PROGRAM Main2
VAR	
	Sequence2 				: Sequence2;
	Reset2					: FB_ResetAllAxis;
	fbStopAll				: FB_StopAll;
	fbPowerAll				: FB_PowerAll;
	bSequenceExecute		: BOOL;
	bUserIncrementStep		: BOOL;
	bUserInfiniteMovement	: BOOL;
	bResetExecute			: BOOL;
	MainState 				: MainStateAxis_enum;
	mainCommands			: MainCommands_typ;
	XYParamaters			: XYParams_typ;
	
	bStopAll: BOOL;
	bPowerEnable: BOOL;
	
	//Test Variables
	
	
	{attribute 'instance-path'}
	{attribute 'no-init'}
	InstancePath			: STRING;
	btest: BOOL;
	AirVariable				AT %Q* : BOOL;
	
	internalEnable			: BOOL;
	internalDisable			: BOOL;
	
	//internalCurrentMoveType	: DeltaCommandType_enum;
	
	internalState			: DeltaState_enum;
	
	internalSetCoordTrafoDone	: BOOL;
	internalMovePathDone		: BOOL;

	
	internalInitObjPos		: ARRAY [1..3] OF MC_LREAL := [0,0,0];
	internalAxesList		: ST_KinAxes;
	internalCMGroup			: AXES_GROUP_REF;
	
	internalTrackAxis		: REFERENCE TO AXIS_REF;
	
	internalPathBuffer		: ARRAY[0..32767] OF BYTE;
	internalPathData		: MC_PATH_DATA_REF( ADR( internalPathBuffer ), SIZEOF( internalPathBuffer ));
		
	externalRoute			: REFERENCE TO Route;	

	internalActiveCoordRef	: MC_COORD_REF;		

	// Internal function blocks
	fbReset_X			: MC_Reset;
	fbReset_Y			: MC_Reset;

	fbPower_X			: MC_Power;
	fbPower_Y			: MC_Power;
	
	fbPower_MCS_X		: MC_Power;
	fbPower_MCS_Y		: MC_Power;
	
	fbAddAxisToGrp			: ARRAY[0..2] OF MC_AddAxisToGroup;
	fbGroupEnable			: MC_GroupEnable;
	
	fbSetCoordTrafo			: MC_SetCoordinateTransform;
	fbMoveLinearPrep		: MC_MoveLinearAbsolutePreparation;
	fbMovePath				: MC_MovePath;
	fbMovePathExt			: MC_MovePath;
	
	//Input Variables
	MotionParameters	: DeltaMotionParameters_typ;			// Motion parameters used by internal motion function blocks	
	myMCSOverride: LREAL := 100.0;
	xSetOverride: BOOL;
	lrGrpOverride: MC_LREAL := 1.0;
	fbMC_GroupSetOverride : MC_GroupSetOverride;
	bTeaching				: BOOL;
	
	//Outputs
	Ready				: BOOL;
	Busy				: BOOL;
	
	Error				: BOOL;
	ErrorID				: UDINT;
	ErrorOrigin			: STRING;
	i: INT;
	
	fbGearIn1:  MC_GearIn;
	bGearIn: BOOL;
END_VAR

(*CASE internalState OF
	DL_IDLE:	// ------------------------------------------------------- idle state
	
		Ready		:= FALSE;
		Busy		:= FALSE;
		
		internalDisable		:= FALSE;
		IF internalEnable THEN
			internalEnable		:= FALSE;
			internalState		:= DL_RESET;
		END_IF
	
	DL_RESET:	// ------------------------------------------------------- resets all axis objects
	
		Ready		:= FALSE;
		Busy		:= TRUE;
		Error		:= FALSE;
		ErrorID		:= 0;
		
		fbReset_X.Execute		:= TRUE;
		fbReset_Y.Execute		:= TRUE;
		
		IF fbReset_X.Done AND
			fbReset_Y.Done THEN
			
			fbReset_X.Execute		:= FALSE;
			fbReset_Y.Execute		:= FALSE;
			
			internalState	:= DL_POWER_AXES;
			
		ELSIF fbReset_X.Error OR
			fbReset_Y.Error THEN
			
			ErrorID; // TODO add whatever the error was for that block
			ErrorOrigin		:= CONCAT( InstancePath, '.fbReset' );
			internalState	:= DL_ERROR; 		
		END_IF
		
	DL_POWER_AXES:	// --------------------------------------------------- energizes all axis objects
	
		Ready		:= FALSE;
		Busy		:= TRUE;
		Error		:= FALSE;
		ErrorID		:= 0;

			fbPower_X.Enable	:= TRUE;
			fbPower_Y.Enable	:= TRUE;

			fbPower_X.Enable_Positive	:= TRUE;
			fbPower_Y.Enable_Positive	:= TRUE;
			
			fbPower_X.Enable_Negative	:= TRUE;
			fbPower_Y.Enable_Negative	:= TRUE;
			
			fbPower_X.Override		:= myMCSOverride;
			fbPower_Y.Override		:= myMCSOverride;
			
			IF fbPower_X.Status AND
				fbPower_Y.Status THEN
				
				internalState	:= DL_ADD_AXES_TO_CM;
				
			ELSIF fbPower_X.Error OR
				fbPower_Y.Error THEN
				
				ErrorID;	// TODO add whatever the error was that block
				ErrorOrigin		:= CONCAT( InstancePath, '.fbPower');
				internalState	:= DL_ERROR;
			END_IF
		
	DL_ADD_AXES_TO_CM:	// ----------------------------------------------- adds MCS axes to CM Group
	
		Ready		:= FALSE;
		Busy		:= TRUE;
		Error		:= FALSE;
		ErrorID		:= 0;

			fbAddAxisToGrp[0].IdentInGroup	:= MCS_X;
			
			fbAddAxisToGrp[1].IdentInGroup	:= MCS_Y;
			
			FOR i := 0 TO 1 DO
				fbAddAxisToGrp[i].Execute		:= TRUE;
			END_FOR
			
			IF fbAddAxisToGrp[0].Done AND
				fbAddAxisToGrp[1].Done THEN
				
				fbAddAxisToGrp[0].Execute	:= FALSE;
				fbAddAxisToGrp[1].Execute	:= FALSE;
				
				internalState	:= DL_ENABLE_CM;
				
			ELSIF fbAddAxisToGrp[0].Error THEN
				fbAddAxisToGrp[0].Execute	:= FALSE;
				fbAddAxisToGrp[1].Execute	:= FALSE;
				
				ErrorID;		// todo : add whichever block errored
				ErrorOrigin		:= CONCAT(InstancePath,'.fbAddAxisToGrp1');
				internalState	:= DL_ERROR;
			ELSIF fbAddAxisToGrp[1].Error THEN
				
				fbAddAxisToGrp[0].Execute	:= FALSE;
				fbAddAxisToGrp[1].Execute	:= FALSE;
				
				ErrorID;		// todo : add whichever block errored
				ErrorOrigin		:= CONCAT(InstancePath,'.fbAddAxisToGrp2');
				internalState	:= DL_ERROR;
			END_IF

	DL_ENABLE_CM:	// ------------------------------------------------------- enables the coordinated motion group
	
		Ready		:= FALSE;
		Busy		:= TRUE;
		Error		:= FALSE;
		ErrorID		:= 0;
		
			fbGroupEnable.Execute		:= TRUE;
			
			IF fbGroupEnable.Done THEN
				internalState	:= DL_RUN;
			ELSIF fbGroupEnable.Error THEN
				ErrorID			:= fbGroupEnable.ErrorId;
				ErrorOrigin		:= CONCAT(InstancePath,'.fbGroupEnable');
				internalState	:= DL_ERROR;
			END_IF
		
	DL_RUN:	// --------------------------------------------------------------- Delta running, ready for commands
	
		Ready		:= TRUE;
		Busy		:= FALSE;
		Error		:= FALSE;
		ErrorID		:= 0;
				
		// reset all commanded function blocks when the execute is recieved
		IF fbSetCoordTrafo.Busy OR fbSetCoordtrafo.CommandAborted THEN
			fbSetCoordTrafo.Execute		:= FALSE;
		ELSIF fbMovePath.Busy OR fbMovePath.CommandAborted THEN
			fbMovePath.Execute			:= FALSE;
		ELSIF fbMovePathEXT.Busy OR fbMovePathEXT.CommandAborted THEN
			fbMovePath.Execute			:= FALSE;
		END_IF
		
		// and catch all internal function block errors
		IF fbSetCoordTrafo.Error THEN
			ErrorID			:= fbSetCoordTrafo.ErrorId;
			ErrorOrigin		:= CONCAT( InstancePath, '.fbSetCoordTrafo' );
			internalState	:= DL_ERROR;
		ELSIF fbMovePath.Error THEN
			ErrorID			:= fbMovePath.ErrorId;
			ErrorOrigin		:= CONCAT( InstancePath, '.fbMovePath' );
			internalState	:= DL_ERROR;
		ELSIF fbMovePathEXT.Error THEN
			ErrorID			:= fbMovePathEXT.ErrorId;
			ErrorOrigin		:= CONCAT( InstancePath, '.fbMovePathEXT' );
			internalState	:= DL_ERROR;
		END_IF
	
	DL_ERROR:	// ----------------------------------------------------------- Error state
	
		Ready		:= FALSE;
		Busy		:= FALSE;
		Error		:= TRUE;
	
END_CASE

fbReset_X( Axis := GVL_XY.stAxis[1] );
fbReset_Y( Axis := GVL_XY.stAxis[2] );

fbPower_X( Axis := GVL_XY.stAxis[1] );
fbPower_Y( Axis := GVL_XY.stAxis[2] );

(*fbPower_MCS_X( Axis := GVL_XY.stAxis[1] );
fbPower_MCS_Y( Axis := GVL_XY.stAxis[2] );*)

fbAddAxisToGrp[0]( AxesGroup := internalCMGroup, Axis := GVL_XY.stAxis[1] );
fbAddAxisToGrp[1]( AxesGroup := internalCMGroup, Axis := GVL_XY.stAxis[2] );

fbGroupEnable( AxesGroup := internalCMGroup );

fbSetCoordTrafo( AxesGroup := internalCMGroup );

fbMovePath( AxesGroup := internalCMGroup, PathData := internalPathData );
fbMovePathEXT( AxesGroup := internalCMGroup, PathData := externalRoute.PathData );

fbMC_GroupSetOverride(
	AxesGroup:= internalCMGroup, 
	Enable:= xSetOverride, 
	VelFactor:= lrGrpOverride, 
	Enabled=> , 
	Busy=> , 
	Error=> , 
	ErrorId=> , 
	ActualVelFactor=> );
	
fbGearIn1(
	Master:= GVL_XY.stAxis[1], 
	Slave:= GVL_XY.stSlaveAxis[1], 
	Execute:= bGearIn, 
	RatioNumerator:= 1, 
	RatioDenominator:= 1, 
	Acceleration:= , 
	Deceleration:= , 
	Jerk:= , 
	BufferMode:= , 
	Options:= , 
	InGear=> , 
	Busy=> , 
	Active=> , 
	CommandAborted=> , 
	Error=> , 
	ErrorID=> );
	
	*)
Sequence2(
	Execute := bSequenceExecute,
	bUserIncrementStep := XYParamaters.bUserIncrementStep,
	bUserInfiniteMovement := XYParamaters.bUserInfiniteMovement,
);

fbPowerAll(
	Enable := bPowerEnable
	);

Reset2(
	Execute := bResetExecute
	);
	
fbStopAll(
		Execute := bStopAll
		);

CASE MainState OF
	
	MSA_DISABLED:
		mainCommands.Start := FALSE;
		mainCommands.Stop := FALSE;
		
	IF mainCommands.Enable THEN
		mainCommands.Disable := FALSE;
		mainState := MSA_INITIALIZING;
	END_IF
		
	MSA_INITIALIZING:
		XYParamaters.bUserIncrementStep := FALSE;
		XYParamaters.bUserInfiniteMovement := TRUE;
		XYParamaters.fVelFactor := 1.0;
		
		IF MainCommands.Disable THEN
			MainCommands.Enable		:=FALSE;
			MainState:= MS_DISABLED;
		ELSIF MainCommands.Stop THEN
			MainCommands.Stop		:=FALSE;
			MainCommands.Disable	:=TRUE;
			MainCommands.Start		:=FALSE;
			MainState	:= MS_DISABLED;
		ELSIF MainCommands.Enable THEN
        	MainState 	:= MSA_ENABLING;
		END_IF
		
	MSA_ENABLING:
		bResetExecute := TRUE;
			IF MainCommands.Disable THEN
				MainCommands.Enable		:=FALSE;
            	MainState	:= MSA_DISABLED;
			ELSIF MainCommands.Stop	 THEN
				MainCommands.Start		:=FALSE;
				MainState	:= MSA_STOPPING;
			ELSIF MainCommands.Enable THEN
				IF Reset2.Done THEN
					bResetExecute := FALSE;
					bPowerEnable := TRUE;
					IF fbPowerAll.Done THEN
						bPowerEnable := FALSE;
						MainState 	:= MSA_ENABLED;
					END_IF	
				END_IF	
			END_IF

	MSA_ENABLED:
		
		MainCommands.Stop := FALSE;
		
		IF MainCommands.Start THEN
			MainState := MSA_RUN;
		ELSIF MainCommands.Disable THEN
            MainCommands.Enable := FALSE;
            MainState           := MSA_STOPPING;
        END_IF
			
	MSA_RUN:
		bSequenceExecute := TRUE;
		
		IF Sequence2.Error THEN
			MainState := MSA_STOPPING;
		END_IF
		
		IF MainCommands.Stop THEN
            MainCommands.Start := FALSE;
            MainState          := MSA_STOPPING;
        ELSIF MainCommands.Disable THEN
            MainCommands.Enable := FALSE;
            MainState           := MSA_STOPPING;
        END_IF
		
	MSA_STOPPING:
		bUserInfiniteMovement := FALSE;
		bUserIncrementStep := FALSE;
		bSequenceExecute := FALSE;
		
		bStopAll := TRUE;
		
		IF fbStopAll.Done THEN
			MainState := MSA_STOPPED;
		END_IF
		
	MSA_STOPPED:
		IF MainCommands.Disable THEN
            MainCommands.Enable := FALSE;
			MainCommands.Start:=FALSE;
            MainState           := MSA_DISABLING;
        ELSIF MainCommands.Start THEN
            MainCommands.Stop := FALSE;
            MainState         := MSA_ENABLING;
        END_IF
		
	MSA_DISABLING:
		bPowerEnable := FALSE;
		bUserIncrementStep := TRUE;
			bUserIncrementStep := FALSE;
			bSequenceExecute := FALSE;
			
			bStopAll := TRUE;
			
			IF fbStopAll.Done THEN
				bStopAll := FALSE;
				MainState := MSA_DISABLED;
			END_IF
		
END_CASE

END_PROGRAM

(* stored: Version 1.1.0.1, ProductVersion 3.1.4024.11
   POU Main2: Id {cef6c1f9-2a01-4b71-81db-f7ed4deb6965}, SpecialFunc None *)
